// TIA Portal V18 export
DATA_BLOCK "OAT"   // DB98
{ S7_Optimized_Access := 'FALSE' }
VERSION : 0.1
// stored: AutoNumber false, DBAccessibleFromOPCUA true, IsOnlyStoredInLoadMemory false, IsWriteProtectedInAS false
   VAR
      Temp { S7_SetPoint := 'True'} : "UDT_OAT";
      cSelectOATMode { S7_SetPoint := 'True'} : Byte;
   END_VAR
BEGIN
END_DATA_BLOCK
